(* CoDeSys 2.3.9.415 project: A1.pro *)
(* Libraries: STANDARD.LIB 15.6.21 11:37:35, IECSFC.LIB 15.6.21 11:37:35, SYSLIBTIME.LIB 18.6.21 10:30:26, SYSTASKINFO.LIB 18.6.21 10:30:26, ANALYZATION.LIB 15.6.21 11:37:35, SYSLIBCALLBACK.LIB 18.6.21 10:30:26 *)

(* PLC configuration (modules and I/O channels)
DI AT %IB0.0 [ByteInput] 8 discrete inputs
Discrete output 2 bit [ID101] node 1, in %IB1 out %QB1 {PinCount = 2; SafeValueBool = FALSE; SafeValueBool = FALSE; Visibility = No}
  AT %QX1.0 [BitOutput] First
  AT %QX1.1 [BitOutput] Second
Discrete output 2 bit [ID101] node 2, in %IB2 out %QB2 {PinCount = 2; SafeValueBool = FALSE; SafeValueBool = FALSE; Visibility = No}
  AT %QX2.0 [BitOutput] First
  AT %QX2.1 [BitOutput] Second
Discrete output 2 bit [ID101] node 3, in %IB3 out %QB3 {PinCount = 2; SafeValueBool = FALSE; SafeValueBool = FALSE; Visibility = No}
  AT %QX3.0 [BitOutput] First
  AT %QX3.1 [BitOutput] Second
Discrete output 2 bit [ID101] node 4, in %IB4 out %QB4 {PinCount = 2; SafeValueBool = FALSE; SafeValueBool = FALSE; Visibility = No}
  AT %QX4.0 [BitOutput] First
  AT %QX4.1 [BitOutput] Second
Discrete output 2 bit [ID101] node 5, in %IB5 out %QB5 {PinCount = 2; SafeValueBool = FALSE; SafeValueBool = FALSE; Visibility = No}
  AT %QX5.0 [BitOutput] First
  AT %QX5.1 [BitOutput] Second
Discrete output 2 bit [ID101] node 6, in %IB6 out %QB6 {PinCount = 2; SafeValueBool = FALSE; SafeValueBool = FALSE; Visibility = No}
  AT %QX6.0 [BitOutput] First
  AT %QX6.1 [BitOutput] Second
Special output [ID104] node 7, in %IB7 out %QB7 {Visibility = No; PinCount = 1}
  AT %QX7.0 [BitOutput] Special output
*)
